PROGRAM main
VAR
    Enable AT %QX0.0 : BOOL;
    ResetTimer AT %QX0.1 : BOOL;
    Done AT %QX0.2 : BOOL;

    RetentiveTimer : TF_RTO;
    Preset : TIME := T#5s;
    ElapsedTime : TIME;
    ElapsedSeconds AT %MD0 : DINT;
    TimerEnabled AT %QX0.3 : BOOL;
    TimerTiming AT %QX0.4 : BOOL;
END_VAR

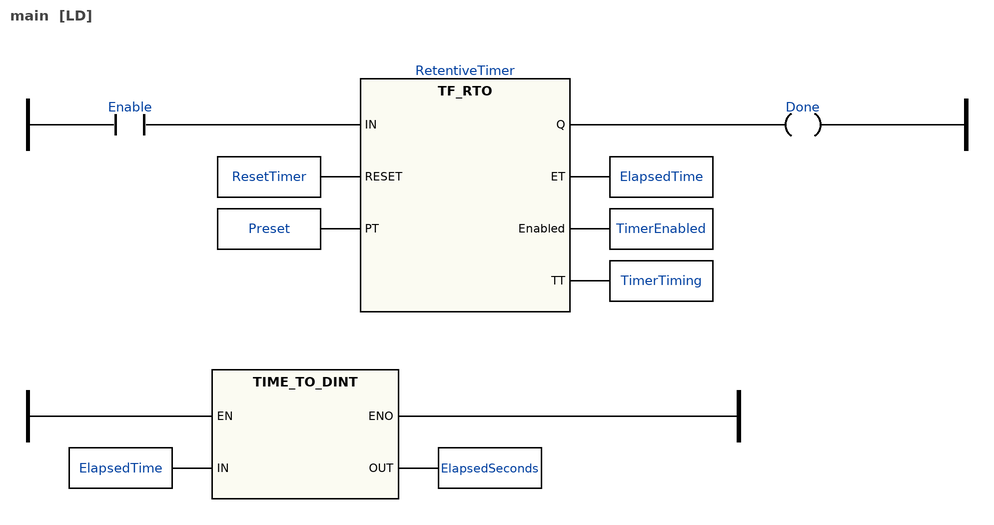
(* LD diagram, written out as Structured Text *)
RetentiveTimer(IN := Enable, RESET := ResetTimer, PT := Preset);
Done := RetentiveTimer.Q;
ElapsedTime := RetentiveTimer.ET;
TimerEnabled := RetentiveTimer.Enabled;
TimerTiming := RetentiveTimer.TT;
ElapsedSeconds := TIME_TO_DINT(ElapsedTime);
END_PROGRAM
